TYPE Gate_Station_DUT :
STRUCT
	Requested_Access:	BOOL;
	Secure_Access:	BOOL;
	Safe_To_Restart:	BOOL;
END_STRUCT
END_TYPE

(* stored: Version 1.1.0.1
   DUT Gate_Station_DUT: Id {3c20b5de-d519-4ce3-b623-7e1ffca0404e} *)
